{attribute 'qualified_only'}
{attribute 'strict'}
TYPE L_Apertures :
(
    SL1L0 := 1,
    SL2L0 := 2
);
END_TYPE

(* stored: Version 1.1.0.1, ProductVersion 3.1.4022.18
   EnumerationTextList L_Apertures: Id {894d4fff-bd3f-4ef2-a8fa-499ec344c700} *)
